// TIA Portal V19 export
VAR_GLOBAL   // PLC tag table "Default tag table"
   System_Byte AT %MB1 : Byte;
   FirstScan AT %M1.0 : Bool;
   DiagStatusUpdate AT %M1.1 : Bool;
   AlwaysTRUE AT %M1.2 : Bool;
   AlwaysFALSE AT %M1.3 : Bool;
   Clock_Byte AT %MB0 : Byte;
   Clock_10Hz AT %M0.0 : Bool;
   Clock_5Hz AT %M0.1 : Bool;
   "Clock_2.5Hz" AT %M0.2 : Bool;
   Clock_2Hz AT %M0.3 : Bool;
   "Clock_1.25Hz" AT %M0.4 : Bool;
   Clock_1Hz AT %M0.5 : Bool;
   "Clock_0.625Hz" AT %M0.6 : Bool;
   "Clock_0.5Hz" AT %M0.7 : Bool;
   Emergency_Stop_OK AT %M52.2 : Bool;
   Emergency_Stop_Status_150K1 AT %I1.0 : Bool;
   Sensor_102B2 AT %I1.1 : Bool;
   Sensor_102B3 AT %I1.2 : Bool;
   Sensor_102B4 AT %I1.3 : Bool;
   Sensor_102B5 AT %I1.4 : Bool;
   Sensor_102B6 AT %I1.5 : Bool;
   Valve_106Q6 AT %Q1.0 : Bool;
   Motor_4Q3 AT %Q1.1 : Bool;
   Motor_4Q5 AT %Q1.2 : Bool;
   Motor_6Q1 AT %Q1.3 : Bool;
   Motor_6Q3 AT %Q1.4 : Bool;
   Reset_Safety_150K1 AT %Q1.5 : Bool;
   HMI_Start AT %M51.6 : Bool;
   HMI_Pause AT %M51.7 : Bool;
   HMI_Reset AT %M52.0 : Bool;
END_VAR
